(* PLC project TEST.project, CODESYS CODESYS V3.5 SP3 Patch 7 *)
(* stored: creationDateTime 2013-12-18T19:57:22.6611883, modificationDateTime 2013-12-18T19:56:09.7450178 *)

FUNCTION_BLOCK Sensor
  VAR
    Induktionsstrom : BOOL;
    ENDE : BOOL;
  END_VAR

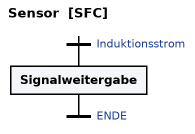
INITIAL_STEP  Sensor bereit:
END_STEP
TRANSITION FROM  Sensor bereit TO Signalweitergabe
  := Induktionsstrom;
END_TRANSITION
STEP Signalweitergabe:
END_STEP
TRANSITION FROM Signalweitergabe TO Init
  := ENDE;
END_TRANSITION
END_FUNCTION_BLOCK
